FUNCTION_BLOCK ABSTRACT FB_Actor2Point
VAR_INPUT
	bSetStatusOnAutomatic : BOOL; //turn actor on
	bAlgorithmPermission : BOOL; //is true if control by algorithm is allowed
END_VAR
VAR_OUTPUT
	bStatusOn : BOOL;
END_VAR
VAR
	{attribute 'OPC.UA.DA' := '1'}
	control : ST_Control;
	{attribute 'OPC.UA.DA' := '1'}
	controlState : ST_ControlState;

	//internal variables
	bSetStatusOn : BOOL; //actual internal value to switch on 
END_VAR

bStatusOn := controlState.bStatusOn;

METHOD PROTECTED SelectControlMode : BOOL
VAR_INPUT
END_VAR

VAR
END_VAR
//change access mode
IF control.bManualModeActivated THEN
	controlState.nAccessmode := E_SystemControlState.manual;
	controlState.sAccessMode := 'manual';
	bSetStatusOn := control.bSetStatusOnManual;
ELSIF control.bAlgorithmModeActivated AND bAlgorithmPermission THEN
	controlState.nAccessmode := E_SystemControlState.algorithm;
	controlState.sAccessMode := 'algorithm';
	bSetStatusOn := control.bSetStatusOnAlgorithm;
ELSE
	controlState.nAccessmode := E_SystemControlState.automatic;
	controlState.sAccessMode := 'automatic';
	bSetStatusOn := bSetStatusOnAutomatic;
END_IF
END_METHOD

END_FUNCTION_BLOCK

(* stored: Version 1.1.0.1, ProductVersion 3.1.4024.9
   POU FB_Actor2Point: Id {779c39b8-c120-47da-8edf-760811555f3b}, SpecialFunc None
   Method SelectControlMode: Id {3e578076-f21b-4cb6-b8d9-37cde3c10288} *)
